TYPE ST_SkillSpecific :
STRUCT
END_STRUCT
END_TYPE

(* stored: Version 1.1.0.1, ProductVersion 3.1.4026.18
   DUT ST_SkillSpecific: Id {9d5d54fc-4f36-486a-9d2e-dbedf970f03f} *)
